FUNCTION_BLOCK FB_PeristalticPump EXTENDS FB_AnalyticalDevices
VAR_INPUT
END_VAR
VAR_OUTPUT
END_VAR
VAR
END_VAR

METHOD TriggerPumpOff : BOOL
VAR_INPUT
END_VAR
END_METHOD

METHOD TriggerPumpOn : BOOL
VAR_INPUT
END_VAR
END_METHOD

END_FUNCTION_BLOCK

(* stored: Version 1.1.0.1
   POU FB_PeristalticPump: Id {6a98df46-caea-4a8a-a9c8-9436707488f6}, SpecialFunc None
   Method TriggerPumpOff: Id {fda3337d-a54d-4819-bd4c-1e4f5f640540}
   Method TriggerPumpOn: Id {87cc8a40-452c-41b4-97a7-da175f8d52c4} *)
